DATA_BLOCK "DB_HBO_Type"
TITLE =%version: 0.05 % CN: 20
//History:
//This version  %created_by: nldy %
//              %date_created: Tuesday, June 06, 2017 10:20:45 AM %
//              %release: VI_GEN/RA_Dev %
//
//Modification History:                                   By:      Date:   Rev:
//----------------------------------------------------  -------  --------  -----
//ra#22220: Update to latest PDB & IDD                   nldy    06-06-17  0.05
//ra#22220: Add gantry motor fault                       nldy    19-04-17  0.04
//ra#21036: Set -1 for unused statuses                   nldy    13-03-17  0.03
//ra#21036: Development + Move to GEN                    nldy    06-03-17  0.02
//Initial version                                        nldy    15-11-16  0.01
//
FAMILY : General
VERSION : 0.0


  STRUCT
   Type_Component : BYTE ;	//Type of the component (1 = Section, 0 = Other)
   Record_Length : BYTE ;	//Number of the Detailed Status in the UDT
   Status : ARRAY  [1 .. 32 ] OF "UDT_Comp_Status";
  END_STRUCT ;
BEGIN
   Type_Component := B#16#0;
   Record_Length := B#16#32;
   Status[1].HMI_Text_Number := 210;
   Status[1].Overall_Status_Relation := B#16#4;
   Status[1].General_Status_Relation := B#16#3;
   Status[2].HMI_Text_Number := 211;
   Status[2].Overall_Status_Relation := B#16#4;
   Status[2].General_Status_Relation := B#16#3;
   Status[3].HMI_Text_Number := 51;
   Status[3].Overall_Status_Relation := B#16#4;
   Status[3].General_Status_Relation := B#16#3;
   Status[4].HMI_Text_Number := 140;
   Status[4].Overall_Status_Relation := B#16#5;
   Status[4].General_Status_Relation := B#16#4;
   Status[5].HMI_Text_Number := 341;
   Status[5].Overall_Status_Relation := B#16#2;
   Status[5].General_Status_Relation := B#16#2;
   Status[6].HMI_Text_Number := 335;
   Status[6].Overall_Status_Relation := B#16#5;
   Status[6].General_Status_Relation := B#16#4;
   Status[7].HMI_Text_Number := 336;
   Status[7].Overall_Status_Relation := B#16#5;
   Status[7].General_Status_Relation := B#16#4;
   Status[8].HMI_Text_Number := 344;
   Status[8].Overall_Status_Relation := B#16#5;
   Status[8].General_Status_Relation := B#16#4;
   Status[9].HMI_Text_Number := -1;
   Status[9].Overall_Status_Relation := B#16#0;
   Status[9].General_Status_Relation := B#16#0;
   Status[10].HMI_Text_Number := -1;
   Status[10].Overall_Status_Relation := B#16#0;
   Status[10].General_Status_Relation := B#16#0;
   Status[11].HMI_Text_Number := -1;
   Status[11].Overall_Status_Relation := B#16#0;
   Status[11].General_Status_Relation := B#16#0;
   Status[12].HMI_Text_Number := -1;
   Status[12].Overall_Status_Relation := B#16#0;
   Status[12].General_Status_Relation := B#16#0;
   Status[13].HMI_Text_Number := -1;
   Status[13].Overall_Status_Relation := B#16#0;
   Status[13].General_Status_Relation := B#16#0;
   Status[14].HMI_Text_Number := 137;
   Status[14].Overall_Status_Relation := B#16#2;
   Status[14].General_Status_Relation := B#16#2;
   Status[15].HMI_Text_Number := 337;
   Status[15].Overall_Status_Relation := B#16#5;
   Status[15].General_Status_Relation := B#16#4;
   Status[16].HMI_Text_Number := 334;
   Status[16].Overall_Status_Relation := B#16#2;
   Status[16].General_Status_Relation := B#16#2;
   Status[17].HMI_Text_Number := 149;
   Status[17].Overall_Status_Relation := B#16#4;
   Status[17].General_Status_Relation := B#16#3;
   Status[18].HMI_Text_Number := 49;
   Status[18].Overall_Status_Relation := B#16#4;
   Status[18].General_Status_Relation := B#16#3;
   Status[19].HMI_Text_Number := 29;
   Status[19].Overall_Status_Relation := B#16#4;
   Status[19].General_Status_Relation := B#16#3;
   Status[20].HMI_Text_Number := 338;
   Status[20].Overall_Status_Relation := B#16#4;
   Status[20].General_Status_Relation := B#16#3;
   Status[21].HMI_Text_Number := 343;
   Status[21].Overall_Status_Relation := B#16#4;
   Status[21].General_Status_Relation := B#16#3;
   Status[22].HMI_Text_Number := -1;
   Status[22].Overall_Status_Relation := B#16#0;
   Status[22].General_Status_Relation := B#16#0;
   Status[23].HMI_Text_Number := 345;
   Status[23].Overall_Status_Relation := B#16#4;
   Status[23].General_Status_Relation := B#16#3;
   Status[24].HMI_Text_Number := 16;
   Status[24].Overall_Status_Relation := B#16#4;
   Status[24].General_Status_Relation := B#16#3;
   Status[25].HMI_Text_Number := 346;
   Status[25].Overall_Status_Relation := B#16#4;
   Status[25].General_Status_Relation := B#16#3;
   Status[26].HMI_Text_Number := 347;
   Status[26].Overall_Status_Relation := B#16#4;
   Status[26].General_Status_Relation := B#16#3;
   Status[27].HMI_Text_Number := 66;
   Status[27].Overall_Status_Relation := B#16#4;
   Status[27].General_Status_Relation := B#16#3;
   Status[28].HMI_Text_Number := 67;
   Status[28].Overall_Status_Relation := B#16#4;
   Status[28].General_Status_Relation := B#16#3;
   Status[29].HMI_Text_Number := 50;
   Status[29].Overall_Status_Relation := B#16#5;
   Status[29].General_Status_Relation := B#16#4;
   Status[30].HMI_Text_Number := -1;
   Status[30].Overall_Status_Relation := B#16#0;
   Status[30].General_Status_Relation := B#16#0;
   Status[31].HMI_Text_Number := -1;
   Status[31].Overall_Status_Relation := B#16#0;
   Status[31].General_Status_Relation := B#16#0;
   Status[32].HMI_Text_Number := -1;
   Status[32].Overall_Status_Relation := B#16#0;
   Status[32].General_Status_Relation := B#16#0;
END_DATA_BLOCK

